# EPICS autosave request: ipApp/Db/Protura_P201_settings.req
$(P)$(ENC)RBV.SCAN
$(P)$(ENC)Pos.ESLO
$(P)$(ENC)Pos.EGU
$(P)$(ENC)Pos.PREC
$(P)$(ENC)Pos.EOFF
